(* IEC 61131-3 sources: PLC-GroupProject/UAS_PLC/build, 2 files *)

(* ---- plc.st ---- *)
TYPE
  LOGLEVEL : (CRITICAL, WARNING, INFO, DEBUG) := INFO;
END_TYPE

FUNCTION_BLOCK LOGGER
  VAR_INPUT
    TRIG : BOOL;
    MSG : STRING;
    LEVEL : LOGLEVEL := INFO;
  END_VAR
  VAR
    TRIG0 : BOOL;
  END_VAR

  IF TRIG AND NOT TRIG0 THEN
  {{
   LogMessage(GetFbVar(LEVEL),(char*)GetFbVar(MSG, .body),GetFbVar(MSG, .len));
  }}
  END_IF;
  TRIG0:=TRIG;
END_FUNCTION_BLOCK

FUNCTION_BLOCK python_eval
  VAR_INPUT
    TRIG : BOOL;
    CODE : STRING;
  END_VAR
  VAR_OUTPUT
    ACK : BOOL;
    RESULT : STRING;
  END_VAR
  VAR
    STATE : DWORD;
    BUFFER : STRING;
    PREBUFFER : STRING;
    TRIGM1 : BOOL;
    TRIGGED : BOOL;
  END_VAR

  {extern void __PythonEvalFB(int, PYTHON_EVAL*);__PythonEvalFB(0, data__);}
END_FUNCTION_BLOCK

FUNCTION_BLOCK python_poll
  VAR_INPUT
    TRIG : BOOL;
    CODE : STRING;
  END_VAR
  VAR_OUTPUT
    ACK : BOOL;
    RESULT : STRING;
  END_VAR
  VAR
    STATE : DWORD;
    BUFFER : STRING;
    PREBUFFER : STRING;
    TRIGM1 : BOOL;
    TRIGGED : BOOL;
  END_VAR

  {extern void __PythonEvalFB(int, PYTHON_EVAL*);__PythonEvalFB(1,(PYTHON_EVAL*)(void*)data__);}
END_FUNCTION_BLOCK

FUNCTION_BLOCK python_gear
  VAR_INPUT
    N : UINT;
    TRIG : BOOL;
    CODE : STRING;
  END_VAR
  VAR_OUTPUT
    ACK : BOOL;
    RESULT : STRING;
  END_VAR
  VAR
    py_eval : python_eval;
    COUNTER : UINT;
    _TMP_ADD10_OUT : UINT;
    _TMP_EQ13_OUT : BOOL;
    _TMP_SEL15_OUT : UINT;
    _TMP_AND7_OUT : BOOL;
  END_VAR

  _TMP_ADD10_OUT := ADD(COUNTER, 1);
  _TMP_EQ13_OUT := EQ(N, _TMP_ADD10_OUT);
  _TMP_SEL15_OUT := SEL(_TMP_EQ13_OUT, _TMP_ADD10_OUT, 0);
  COUNTER := _TMP_SEL15_OUT;
  _TMP_AND7_OUT := AND(_TMP_EQ13_OUT, TRIG);
  py_eval(TRIG := _TMP_AND7_OUT, CODE := CODE);
  ACK := py_eval.ACK;
  RESULT := py_eval.RESULT;
END_FUNCTION_BLOCK

PROGRAM UAS_PLC
  VAR
    START : BOOL;
    STOP : BOOL;
    CR_MOTOR1 : BOOL;
    MOTOR_PUMP1 : BOOL;
    LEVEL_SWITCH2 : BOOL;
    LEVEL_SWITCH1 : BOOL;
    CR_LEVEL1 : BOOL;
    CR_LEVEL2 : BOOL;
    PL1 : BOOL;
    PL2 : BOOL;
    CR1 : BOOL;
    CR2 : BOOL;
    SOLENOID_VALVE1 : BOOL;
    SOLENOID_VALVE2 : BOOL;
  END_VAR

  CR_MOTOR1 := NOT(CR_LEVEL2) AND NOT(STOP) AND (CR_MOTOR1 OR START);
  MOTOR_PUMP1 := CR_MOTOR1;
  CR1 := NOT(CR_LEVEL1) AND CR_MOTOR1;
  SOLENOID_VALVE1 := CR1;
  CR_LEVEL1 := LEVEL_SWITCH1;
  CR2 := NOT(CR_LEVEL2) AND CR_LEVEL1 AND CR_MOTOR1;
  SOLENOID_VALVE2 := CR2;
  CR_LEVEL2 := LEVEL_SWITCH2;
  PL1 := CR_LEVEL1;
  PL2 := CR_LEVEL2;
END_PROGRAM

CONFIGURATION Config0

  RESOURCE Res0 ON PLC
    TASK task0(INTERVAL := T#20ms,PRIORITY := 0);
    PROGRAM instance0 WITH task0 : UAS_PLC;
  END_RESOURCE
END_CONFIGURATION

(* ---- generated_plc.st ---- *)
PROGRAM UAS_PLC
  VAR
    START : BOOL;
    STOP : BOOL;
    CR_MOTOR1 : BOOL;
    MOTOR_PUMP1 : BOOL;
    LEVEL_SWITCH2 : BOOL;
    LEVEL_SWITCH1 : BOOL;
    CR_LEVEL1 : BOOL;
    CR_LEVEL2 : BOOL;
    PL1 : BOOL;
    PL2 : BOOL;
    CR1 : BOOL;
    CR2 : BOOL;
    SOLENOID_VALVE1 : BOOL;
    SOLENOID_VALVE2 : BOOL;
  END_VAR

  CR_MOTOR1 := NOT(CR_LEVEL2) AND NOT(STOP) AND (CR_MOTOR1 OR START);
  MOTOR_PUMP1 := CR_MOTOR1;
  CR1 := NOT(CR_LEVEL1) AND CR_MOTOR1;
  SOLENOID_VALVE1 := CR1;
  CR_LEVEL1 := LEVEL_SWITCH1;
  CR2 := NOT(CR_LEVEL2) AND CR_LEVEL1 AND CR_MOTOR1;
  SOLENOID_VALVE2 := CR2;
  CR_LEVEL2 := LEVEL_SWITCH2;
  PL1 := CR_LEVEL1;
  PL2 := CR_LEVEL2;
END_PROGRAM

CONFIGURATION Config0

  RESOURCE Res0 ON PLC
    TASK task0(INTERVAL := T#20ms,PRIORITY := 0);
    PROGRAM instance0 WITH task0 : UAS_PLC;
  END_RESOURCE
END_CONFIGURATION
